FUNCTION_BLOCK FB_PositionStatePMPS_Base
(*
    FB_PositionStatePMPS without Arbiter, BPTM, FFO

    This allows me to test most of the code without an arbiter plc setup
*)
VAR_IN_OUT
    stMotionStage: DUT_MotionStage;
    arrStates: ARRAY[1..15] OF DUT_PositionState;
END_VAR
VAR_INPUT
    bRequestTransition: BOOL;
    setState: INT;
    getState: INT;
    fStateBoundaryDeadband: LREAL := 0;
    stTransitionBeam: ST_BeamParams := PMPS_GVL.cstSafeBeam;
    nTransitionAssertionID: UDINT;
END_VAR
VAR_OUTPUT
    bTransitionAuthorized: BOOL;
    bForwardAuthorized: BOOL;
    bBackwardAuthorized: BOOL;
END_VAR
VAR
    bInit: BOOL := TRUE;
    fbLinGov: FB_LinearGovernor;
    rtTransReq: R_TRIG;
    ftTransAuth: F_TRIG;
    stStateReq: DUT_PositionState;
    mcPower: MC_POWER;
    fUpperBound: LREAL;
    fLowerBound: LREAL;
    nGoalState: INT;
    stGoalState: DUT_PositionState;
    fActPos: LREAL;
    fReqPos: LREAL;
    bInTransition: BOOL;
    stBeamNeeded: ST_BeamParams;
END_VAR

// This is meant to be subclassed. The parent class body is in the Exec action.

ACTION Exec:
// Initialize or reinitialize to the current state value
ftTransAuth(CLK:=bTransitionAuthorized);
IF ftTransAuth.Q THEN
    bInit := TRUE;
END_IF
IF bInit THEN
    bInit R= stMotionStage.bAxisParamsInit;
    nGoalState := getState;
    stStateReq := GetStateStruct(getState);
    bInTransition := FALSE;
END_IF

// Request transition on rising edge
rtTransReq(CLK:=bRequestTransition);
IF rtTransReq.Q THEN
    nGoalState := setState;
    stStateReq := GetStateStruct(setState);
    bInTransition := TRUE;
END_IF

// Handles getting the request to the arbiter and back
HandleBPTM();

// Set up MPS virtual limit for moves at and between states
stGoalState := GetStateStruct(nGoalState);
fActPos := stMotionStage.stAxisStatus.fActPosition;
IF stMotionStage.bExecute THEN
    fReqPos := stMotionStage.fPosition;
ELSE
    fReqPos := fActPos;
END_IF

// Start with no move authority
bForwardAuthorized := FALSE;
bBackwardAuthorized := FALSE;

// Grant auth during moves based on goal state, current position, and goal position
IF stMotionStage.bExecute AND stGoalState.bValid THEN
    bForwardAuthorized := F_PosUnderUpperBound(MAX(fActPos, fReqPos) + ABS(fStateBoundaryDeadband), stGoalState);
    bBackwardAuthorized := F_PosOverLowerBound(MIN(fActPos, fReqPos) - ABS(fStateBoundaryDeadband), stGoalState);
END_IF

IF bInTransition THEN
    // Deny auth during a transition request until transition is authorized
    bForwardAuthorized R= NOT bTransitionAuthorized;
    bBackwardAuthorized R= NOT bTransitionAuthorized;
    // Have the motor wait for permission to start move instead of immediately erroring
    stMotionStage.bSafetyReady := bTransitionAuthorized;
ELSE
    // If not transitioning, no need to wait for safety: immediately try to move and error if no auth
    stMotionStage.bSafetyReady := TRUE;
    // Set an error message override in case this causes an error
    IF stMotionStage.bError AND fReqPos > fActPos AND NOT bForwardAuthorized THEN
        stMotionStage.sCustomErrorMessage := 'Unsafe tweak forward blocked by PMPS';
    ELSIF stMotionStage.bError AND fReqPos < fActPos AND NOT bBackwardAuthorized THEN
        stMotionStage.sCustomErrorMessage := 'Unsafe tweak backward blocked by PMPS';
    END_IF
END_IF

// Only let us move if the transition is allowed, or if we are moving within a state's bounds
mcPower(Axis:=stMotionStage.Axis,
        Enable:=stMotionStage.bAllEnable,
        Enable_Positive:=stMotionStage.bAllForwardEnable AND bForwardAuthorized,
        Enable_Negative:=stMotionStage.bAllBackwardEnable AND bBackwardAuthorized);

// Raise fast faults as needed
stBeamNeeded := GetBeamFromState(getState);
HandleFFO();
END_ACTION

METHOD GetBeamFromState : ST_BeamParams;
VAR_INPUT
    nState: INT;
END_VAR
VAR
    stState: DUT_PositionState;
END_VAR
stState := GetStateStruct(nState);
GetBeamFromState := stState.stBeamParams;
END_METHOD

METHOD GetStateCode : INT
VAR_INPUT
    nState: INT;
END_VAR
IF nState < 0 OR nState > 15 THEN
    GetStateCode := -1;
ELSE
    GetStateCode := nState;
END_IF
END_METHOD

METHOD GetStateStruct : DUT_PositionState
VAR_INPUT
    nState: INT;
END_VAR
{warning disable C0371}
// Implicit VAR_IN_OUT reference inside a method needs special handling
IF NOT __ISVALIDREF(arrStates) THEN
    GetStateStruct := MOTION_GVL.stInvalidState;
    RETURN;
END_IF
CASE GetStateCode(nState) OF
    -1: GetStateStruct := MOTION_GVL.stInvalidState;
    0: GetStateStruct := MOTION_GVL.stUnknownState;
    ELSE
        GetStateStruct := arrStates[nState];
END_CASE
{warning restore C0371}
END_METHOD

ACTION HandleBPTM:

END_ACTION

ACTION HandleFFO:

END_ACTION

END_FUNCTION_BLOCK

(* stored: Version 1.1.0.1, ProductVersion 3.1.4022.18
   POU FB_PositionStatePMPS_Base: Id {e35067d1-2ee7-46f4-a240-48505f8439a4}, SpecialFunc None
   Action Exec: Id {5b04393f-c32f-49f1-a610-cb4c89f50675}
   Method GetBeamFromState: Id {ace20d49-ae59-4162-85f5-ab83a2a0552b}
   Method GetStateCode: Id {30e413cd-5f48-49b3-b46d-6cd3e4359ded}
   Method GetStateStruct: Id {fd5be017-4792-4f22-a98a-6c401c8e2c66}
   Action HandleBPTM: Id {b4dce640-f1d3-4191-98dd-b7fe08e15f67}
   Action HandleFFO: Id {4a6d3817-8b4c-48a0-a34b-e22189bbf6e2} *)
